// TIA Portal V16 export
// export: Created 2023-06-21T17:06:26.8199Z, ExportSetting WithDefaults, DisplayName Totally Integrated Automation Portal, DisplayVersion V16 Update 4, DisplayName TIA Portal Version Control Interface, DisplayVersion V16 Update 2, DisplayName TIA Portal Openness, DisplayVersion V16 Update 4, DisplayName SINAMICS Startdrive Advanced, DisplayVersion V16, DisplayName SINAMICS Startdrive G130, G150, S120, S150, SINAMICS MV, S210, DisplayVersion V16, DisplayName SINAMICS Startdrive G110M, G120, G120C, G120D, G120P, DisplayVersion V16, DisplayName STEP 7 Professional, DisplayVersion V16 Update 4, DisplayName STEP 7 Safety, DisplayVersion V16, DisplayName Soft Starter ES, DisplayVersion V16, DisplayName WinCC Advanced, DisplayVersion V16 Update 4
FUNCTION "Word_2_Bool" : Void   // FC1, LAD
{ S7_Optimized_Access := 'TRUE' }
VERSION : 0.1
// stored: AutoNumber true, IsIECCheckEnabled false, SetENOAutomatically false, UDAEnableTagReadback false
   VAR_INPUT
      "1_registrador_in" : Word;
      "2_registrador_in" : Word;
      "3_registrador_in" : Word;
      "4_registrador_in" : Word;
      "5_registrador_in" : Word;
   END_VAR
   VAR_OUTPUT
      Fancoil_Ligado : Bool;
      Heating : Bool;
      Cooling : Bool;
      Fan : Bool;
      Sts_Fan : Bool;
      Sts_Heating : Bool;
      Sts_Cooling : Bool;
      Slave : Bool;
      Master : Bool;
      SP_Out : Real;
      PV_Out : Real;
      Malfunction : Bool;
   END_VAR
   VAR_TEMP
      Aux_1 : Word;
      Aux_2 : Word;
      Aux_3 : Word;
      Aux_4 : Word;
      Temp_Real_Word_1 : Real;
      Temp_Real_Word_2 : Real;
   END_VAR
BEGIN

REGION Network 1: Verifica se esta ligado ou desligado
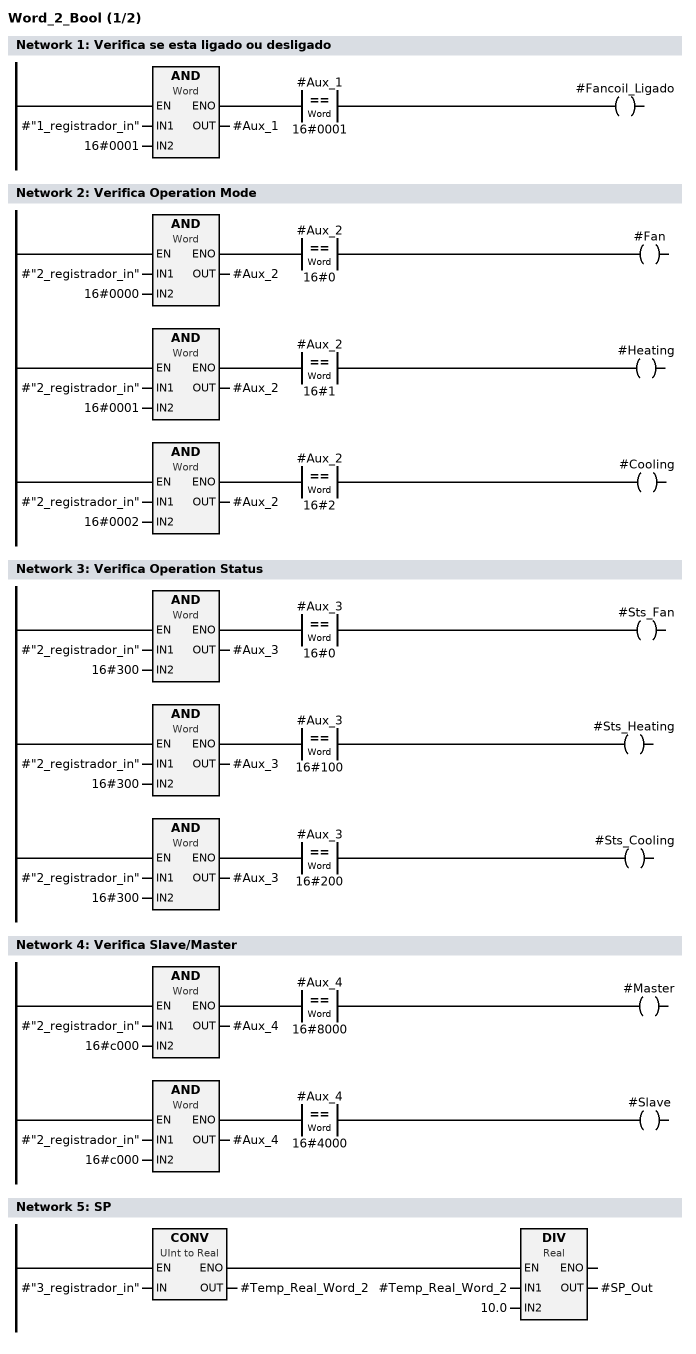
   RUNG wire#powerrail
      { S7_Templates := "SrcType := Word" } And(in1 := #"1_registrador_in", in2 := 16#0001, out => #Aux_1)
      { S7_Templates := "SrcType := Word" } EQ_Contact(in1 := #Aux_1, in2 := 16#0001)
      Coil( #Fancoil_Ligado )
   END_RUNG
   // the same network as SCL:
   #Aux_1 := #"1_registrador_in" AND 16#0001;
   #Fancoil_Ligado := #Aux_1 = 16#0001;
END_REGION

REGION Network 2: Verifica Operation Mode
   RUNG wire#powerrail
      { S7_Templates := "SrcType := Word" } And(in1 := #"2_registrador_in", in2 := 16#0000, out => #Aux_2)
      { S7_Templates := "SrcType := Word" } EQ_Contact(in1 := #Aux_2, in2 := 16#0)
      Coil( #Fan )
   END_RUNG
   RUNG wire#powerrail
      { S7_Templates := "SrcType := Word" } And(in1 := #"2_registrador_in", in2 := 16#0001, out => #Aux_2)
      { S7_Templates := "SrcType := Word" } EQ_Contact(in1 := #Aux_2, in2 := 16#1)
      Coil( #Heating )
   END_RUNG
   RUNG wire#powerrail
      { S7_Templates := "SrcType := Word" } And(in1 := #"2_registrador_in", in2 := 16#0002, out => #Aux_2)
      { S7_Templates := "SrcType := Word" } EQ_Contact(in1 := #Aux_2, in2 := 16#2)
      Coil( #Cooling )
   END_RUNG
   // the same network as SCL:
   #Aux_2 := #"2_registrador_in" AND 16#0000;
   #Fan := #Aux_2 = 16#0;
   #Aux_2 := #"2_registrador_in" AND 16#0001;
   #Heating := #Aux_2 = 16#1;
   #Aux_2 := #"2_registrador_in" AND 16#0002;
   #Cooling := #Aux_2 = 16#2;
END_REGION

REGION Network 3: Verifica Operation Status
   RUNG wire#powerrail
      { S7_Templates := "SrcType := Word" } And(in1 := #"2_registrador_in", in2 := 16#300, out => #Aux_3)
      { S7_Templates := "SrcType := Word" } EQ_Contact(in1 := #Aux_3, in2 := 16#0)
      Coil( #Sts_Fan )
   END_RUNG
   RUNG wire#powerrail
      { S7_Templates := "SrcType := Word" } And(in1 := #"2_registrador_in", in2 := 16#300, out => #Aux_3)
      { S7_Templates := "SrcType := Word" } EQ_Contact(in1 := #Aux_3, in2 := 16#100)
      Coil( #Sts_Heating )
   END_RUNG
   RUNG wire#powerrail
      { S7_Templates := "SrcType := Word" } And(in1 := #"2_registrador_in", in2 := 16#300, out => #Aux_3)
      { S7_Templates := "SrcType := Word" } EQ_Contact(in1 := #Aux_3, in2 := 16#200)
      Coil( #Sts_Cooling )
   END_RUNG
   // the same network as SCL:
   #Aux_3 := #"2_registrador_in" AND 16#300;
   #Sts_Fan := #Aux_3 = 16#0;
   #Aux_3 := #"2_registrador_in" AND 16#300;
   #Sts_Heating := #Aux_3 = 16#100;
   #Aux_3 := #"2_registrador_in" AND 16#300;
   #Sts_Cooling := #Aux_3 = 16#200;
END_REGION

REGION Network 4: Verifica Slave/Master
   RUNG wire#powerrail
      { S7_Templates := "SrcType := Word" } And(in1 := #"2_registrador_in", in2 := 16#c000, out => #Aux_4)
      { S7_Templates := "SrcType := Word" } EQ_Contact(in1 := #Aux_4, in2 := 16#8000)
      Coil( #Master )
   END_RUNG
   RUNG wire#powerrail
      { S7_Templates := "SrcType := Word" } And(in1 := #"2_registrador_in", in2 := 16#c000, out => #Aux_4)
      { S7_Templates := "SrcType := Word" } EQ_Contact(in1 := #Aux_4, in2 := 16#4000)
      Coil( #Slave )
   END_RUNG
   // the same network as SCL:
   #Aux_4 := #"2_registrador_in" AND 16#c000;
   #Master := #Aux_4 = 16#8000;
   #Aux_4 := #"2_registrador_in" AND 16#c000;
   #Slave := #Aux_4 = 16#4000;
END_REGION

REGION Network 5: SP
   RUNG wire#powerrail
      { S7_Templates := "[SrcType := UInt, DestType := Real]" } Convert(in := #"3_registrador_in", out => #Temp_Real_Word_2)
      { S7_Templates := "SrcType := Real" } Div(in1 := #Temp_Real_Word_2, in2 := 10.0, out => #SP_Out)
   END_RUNG
   // the same network as SCL:
   #Temp_Real_Word_2 := UINT_TO_REAL(#"3_registrador_in");
   #SP_Out := #Temp_Real_Word_2 / 10.0;
END_REGION

REGION Network 6: PV
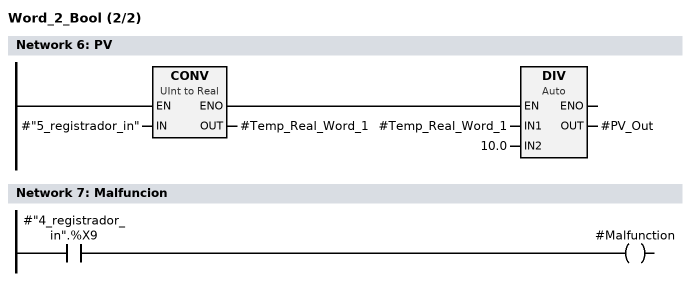
   RUNG wire#powerrail
      { S7_Templates := "[SrcType := UInt, DestType := Real]" } Convert(in := #"5_registrador_in", out => #Temp_Real_Word_1)
      Div(in1 := #Temp_Real_Word_1, in2 := 10.0, out => #PV_Out)
   END_RUNG
   // the same network as SCL:
   #Temp_Real_Word_1 := UINT_TO_REAL(#"5_registrador_in");
   #PV_Out := #Temp_Real_Word_1 / 10.0;
END_REGION

REGION Network 7: Malfuncion
   RUNG wire#powerrail
      Contact( #"4_registrador_in".%X9 )
      Coil( #Malfunction )
   END_RUNG
   // the same network as SCL:
   #Malfunction := #"4_registrador_in".%X9;
END_REGION
END_FUNCTION
